# B&R Automation Studio project Prog_3
Automation Studio 4.5.2.102

## Configuration Config1

### Task classes (Cpu.sw)
```
Cyclic#1:
  Program <- Program.prg
Binaries: udbdef, mcacpdrv, arsvcreg, TCData, ashwd, ashwac, asfw, iomap, sysconf, Role, User, arconfig
Libraries: McBase, MpAxis, McAxis, MpBase, McAcpAx, Library, powerlnk, sys_lib, astime, fileio, runtime
```

### Hardware
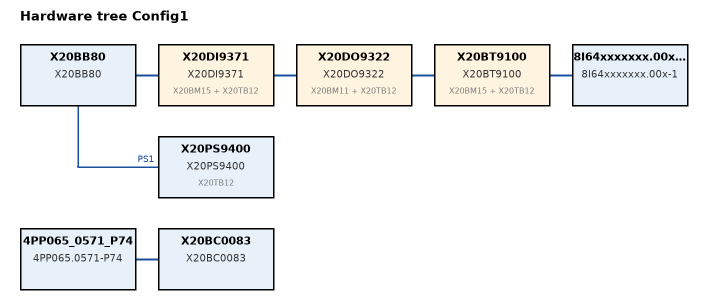
```
4PP065_0571_P74 : 4PP065.0571-P74 v1.1.2.0
  Connector IF5:
    ActivateDevice = 1
    Mode = Manual
    InternetAddress = 10.0.1.10
    SubnetMask = 255.255.255.0
  ConfigurationID = labBR
8I64xxxxxxx.00x-1 : 8I64xxxxxxx.00x-1 v2.1.3.0  [X2X1 -> X20BT9100.X2X1 [Cable Type=X2XCable, Length=10, Version=1.0.0.2]]
  FunctionModel = Standard
  packedETAD = packed
  packedCMDD = packed
X20BB80 : X20BB80 v1.0.2.0
X20BC0083 : X20BC0083 v2.9.0.0  [PLK1 -> 4PP065_0571_P74.IF4 (NodeNumber=2) [Cable Type=PowerlinkCable, Length=10, Version=1.0.0.2]; SL -> X20BB80.SL1]
X20BM11a : X20BM11 v1.0.0.1  [X2X1 -> X20BM15.X2X2]
X20BM15 : X20BM15 v1.0.1.0  [X2X1 -> X20BB80.IF1 (NodeNumber=5)]
X20BM15a : X20BM15 v1.0.1.0  [X2X1 -> X20BM11a.X2X2 (NodeNumber=10)]
X20BT9100 : X20BT9100 v1.0.3.0  [SS1 -> X20TB12f.SS; SL -> X20BM15a.SL1]
X20DI9371 : X20DI9371 v1.0.2.0  [SS1 -> X20TB12a.SS; SL -> X20BM15.SL1]
X20DO9322 : X20DO9322 v1.0.3.0  [SS1 -> X20TB12d.SS; SL -> X20BM11a.SL1]
X20PS9400 : X20PS9400 v1.0.2.4  [SS1 -> X20TB12.SS; PS -> X20BB80.PS1]
X20TB12 : X20TB12 v1.0.0.0
X20TB12a : X20TB12 v1.0.0.0
X20TB12d : X20TB12 v1.0.0.0
X20TB12f : X20TB12 v1.0.0.0
```

### IoMap.iom - 4PP065_0571_P74/IoMap.iom
```iecst
VAR_CONFIG
	::Program:speed AT %QW."8I64xxxxxxx.00x-1".LFRD_Output;
	::Program:servo.STATE AT %IW."8I64xxxxxxx.00x-1".ETAD_Input;
	::Program:servo.COM AT %QW."8I64xxxxxxx.00x-1".CMDD_Output;
	::Program:decrease_speed_btn AT %IX."X20DI9371".DigitalInput02;
	::Program:decrease_speed_btn AT %QX."X20DO9322".DigitalOutput02;
	::Program:on_switch AT %IX."X20DI9371".DigitalInput01;
	::Program:increase_speed_btn AT %IX."X20DI9371".DigitalInput03;
	::Program:increase_speed_btn AT %QX."X20DO9322".DigitalOutput03;
	::Program:reset_btn AT %IX."X20DI9371".DigitalInput04;
	::Program:reset_btn AT %QX."X20DO9322".DigitalOutput04;
	::Program:on_switch AT %QX."X20DO9322".DigitalOutput05;
	::Program:torque AT %IW."8I64xxxxxxx.00x-1".OTR_Input;
END_VAR
```

## Logical view

Binary libraries used (declarations not repeated): operator, runtime, astime, AsIecCon, McBase, MpAxis 5.02.1, McAxis, MpBase, McAcpAx 5.02.1

### Program Logical/Program

#### Variables.var
```iecst
VAR
	speed : INT := 0;
	servo : DRIVE;
	on_switch : BOOL;
	increase_speed_btn : BOOL;
	decrease_speed_btn : BOOL;
	reset_btn : BOOL;
	torque : INT;
	error : BOOL := FALSE;
END_VAR
```

#### Main.c
```c
#include <bur/plctypes.h>

#ifdef _DEFAULT_INCLUDES
	#include <AsDefault.h>
#endif

void _INIT ProgramInit(void) {

}

void _CYCLIC ProgramCyclic(void) {
	if (!error) {
		if (increase_speed_btn && speed < 1000) {
			speed += 1;
		}
		if (decrease_speed_btn && speed > -1000) {
			speed -= 1;
		}
		if (reset_btn) {
			speed = 0;
		}
	}

	if (torque > 6) error = 1;

	if (error && !on_switch) {
		error = 0;
		speed = 0;
	}

	if (!error) {
		servo.ENABLE = on_switch;
	} else {
		servo.ENABLE = 0;
	}

	DRIVE(&servo);
}

void _EXIT ProgramExit(void) {

}
```
